// TIA Portal V17 export
// export: Created 2023-12-22T15:05:34.3097939Z, ExportSetting WithDefaults, DisplayName Totally Integrated Automation Portal, DisplayVersion V17, DisplayName TIA Portal Openness, DisplayVersion V17, DisplayName TIA Portal Version Control Interface, DisplayVersion V17, DisplayName STEP 7 Professional, DisplayVersion V17, DisplayName STEP 7 Safety, DisplayVersion V17, DisplayName WinCC Advanced, DisplayVersion V17
DATA_BLOCK "Logick_DB"   // DB1
VERSION : 0.1
// stored: AutoNumber true, DBAccessibleFromOPCUA true, InstanceOfName Logick, InstanceOfType FB
"Logick"
   // VAR RETAIN
   //    Start_ELZ : Bool;
   //    REQ_Wash : Bool;
   //    Force_Wash : Bool;
   //    ELZ : Bool;
   //    Local : Bool;
   //    Step_Wash : Int;
   //    ELZ_LED : Int;
   //    RM_1 { S7_SetPoint := 'True'} : Real := 0.0;
   //    Alarm : Word;
   //    Alarms : Struct
   //       Gas : Bool;
   //       ELZ_AHLS : Bool;
   //    END_STRUCT;
   //    ELZ_1 { S7_SetPoint := 'True'} : "ELZ";
   //    Days : Struct
   //       D_1 : Bool;
   //       D_2 : Bool;
   //       D_3 : Bool;
   //       D_4 : Bool;
   //       D_5 : Bool;
   //       D_6 : Bool;
   //       D_7 : Bool;
   //    END_STRUCT;
   //    Houres : Struct
   //       H_D_1 : Int;
   //       H_D_2 : Int;
   //       H_D_3 : Int;
   //       H_D_4 : Int;
   //       H_D_5 : Int;
   //       H_D_6 : Int;
   //       H_D_7 : Int;
   //    END_STRUCT;
   //    Minutes : Struct
   //       M_D_1 : Int;
   //       M_D_2 : Int;
   //       M_D_3 : Int;
   //       M_D_4 : Int;
   //       M_D_5 : Int;
   //       M_D_6 : Int;
   //       M_D_7 : Int;
   //    END_STRUCT;
   //    T_Wash { S7_SetPoint := 'True'} : "Time_M";
   // END_VAR
BEGIN
   ELZ_1.T_Gas.SP_M := 0;
   ELZ_1.T_Gas.SP_S := 30;
   ELZ_1.T_ELZ_Start.SP_M := 0;
   ELZ_1.T_ELZ_Start.SP_S := 5;
   T_Wash.SP_M := 0;
   T_Wash.SP_S := 30;
END_DATA_BLOCK
